(* Logix 5000 project; controller Sucrose_Main Emulate 5570 rev 20.12; software revision 20.01; part 10 of 30 *)
(* tags used below, declared in another part *)
   Alarm_ACK_Master_Timer : TIMER;
   DO_E20_6 : ALIAS FOR FLX_E20:6:O;   // Discrete Output EN2T_FLX 192.168.1.20
   DO_E20_7 : ALIAS FOR FLX_E20:7:O;   // Discrete Output EN2T_FLX 192.168.1.20
   DO_E24_3 : ALIAS FOR FLX_E24:3:O;   // Discrete Output EN2T_FLX 192.168.1.24
   FV230103_AOI : QSI_Flow_Valve;   // FV-23-01-03 SUCROSE TANK #1 OUTLET VALVE
   FV230203_AOI : QSI_Flow_Valve;   // FV-23-02-03 SUCROSE TANK #2 OUTLET VALVE
   FV230401_AOI : QSI_Flow_Valve;   // FV-23-04-01 SUCROSE TANK #3 LOW POINT DRAIN
   FV230402_AOI : QSI_Flow_Valve;   // FV-23-04-02 SUCROSE TANK #2 LOW POINT DRAIN
   FV230403_AOI : QSI_Flow_Valve;   // FV-23-04-03 SUCROSE TANK #1 LOW POINT DRAIN
   FV230431_AOI : QSI_Flow_Valve;   // FV-23-04-31 SUCROSE LOW POINT DRAIN VALVE @ TRANSFER PUMP #1
   FV230432_AOI : QSI_Flow_Valve;   // FV-23-04-32 SUCROSE LOW POINT DRAIN VALVE @ TRANSFER PUMP #2
   P230401_AOI : PF525_VFD_E_ENET;   // P-23-04-01 SUCROSE TRANSFER PUMP 1
   P230402_AOI : PF525_VFD_E_ENET;   // P-23-04-02 SUCROSE TRANSFER PUMP 2
   PSV230401_AOI : QSI_Flow_Valve;   // PSV-23-04-01 TRANSFER PUMP #1 BYPASS VALVE
   PSV230402_AOI : QSI_Flow_Valve;   // PSV-23-04-02 TRANSFER PUMP #2 BYPASS VALVE
   Sucrose_MM_Enable : BOOL;
   SucroseCIP_P230401_REMOTE : CIP_REMOTE;
   SucroseCIP_P230402_REMOTE : CIP_REMOTE;
   SucroseCIP_TK230101_REMOTE : CIP_REMOTE;
   SucroseCIP_TK230201_REMOTE : CIP_REMOTE;
   SucroseTanks : Area_Program;
   SV130401_AOI : QSI_Discrete_Device;   // SV-13-04-01 SUCROSE TRANSFER PUMP #1 SEAL WATER FLUSH VALVE
   SV130402_AOI : QSI_Discrete_Device;   // SV-13-04-02 SUCROSE TRANSFER PUMP #2 SEAL WATER FLUSH VALVE
(* DischargeArea_EN2T_IO_Discrete_DO_E20_5, continued *)

ROUTINE MainRoutine   (* ladder *)
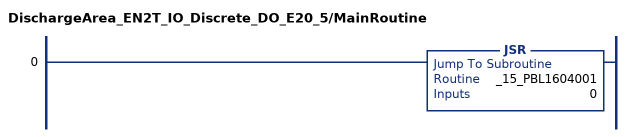
   0: JSR(_15_PBL1604001,0);
END_ROUTINE
END_PROGRAM

PROGRAM DischargeArea_EN2T_IO_Discrete_DO_E20_6   (* main routine MainRoutine *)

ROUTINE _00_FV230431   (* ladder *)
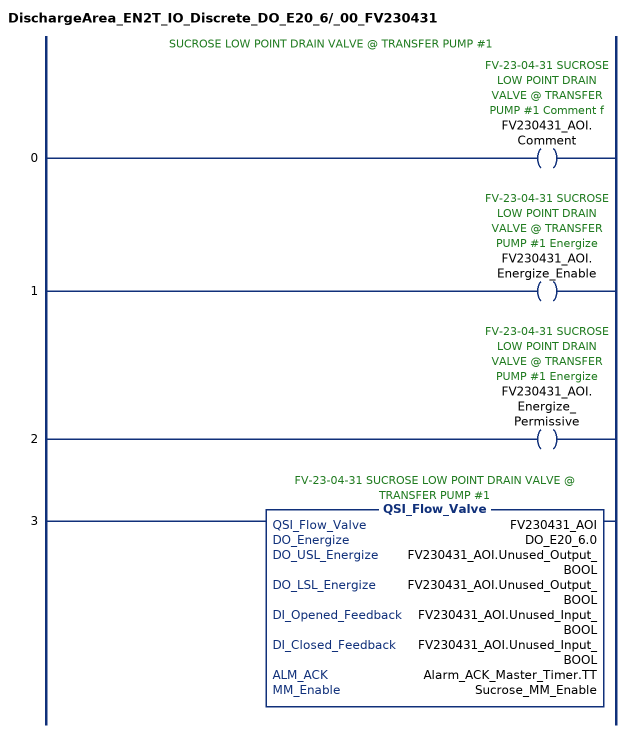
   // SUCROSE LOW POINT DRAIN VALVE @ TRANSFER PUMP #1
   0: OTE(FV230431_AOI.Comment);
   1: OTE(FV230431_AOI.Energize_Enable);
   2: OTE(FV230431_AOI.Energize_Permissive);
   3: QSI_Flow_Valve(FV230431_AOI,DO_E20_6.0,FV230431_AOI.Unused_Output_BOOL,FV230431_AOI.Unused_Output_BOOL,FV230431_AOI.Unused_Input_BOOL,FV230431_AOI.Unused_Input_BOOL,Alarm_ACK_Master_Timer.TT,Sucrose_MM_Enable);
END_ROUTINE

ROUTINE _01_FV230432   (* ladder *)
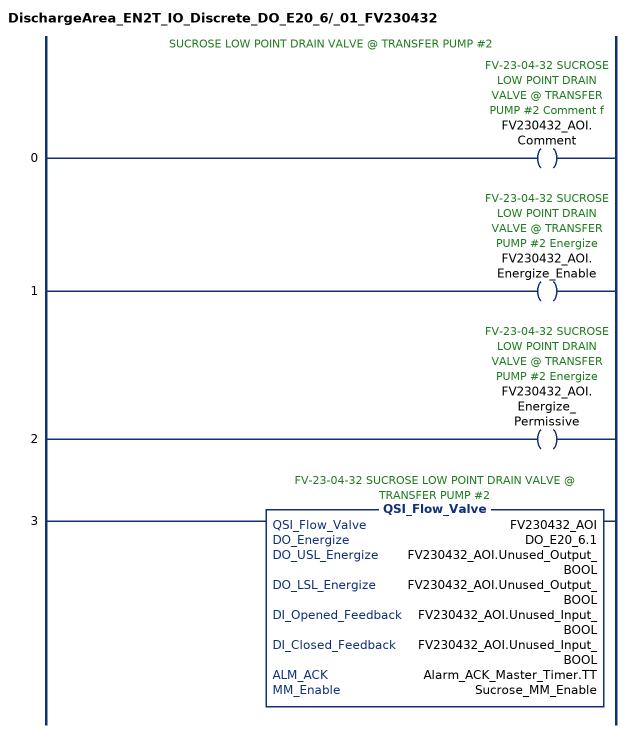
   // SUCROSE LOW POINT DRAIN VALVE @ TRANSFER PUMP #2
   0: OTE(FV230432_AOI.Comment);
   1: OTE(FV230432_AOI.Energize_Enable);
   2: OTE(FV230432_AOI.Energize_Permissive);
   3: QSI_Flow_Valve(FV230432_AOI,DO_E20_6.1,FV230432_AOI.Unused_Output_BOOL,FV230432_AOI.Unused_Output_BOOL,FV230432_AOI.Unused_Input_BOOL,FV230432_AOI.Unused_Input_BOOL,Alarm_ACK_Master_Timer.TT,Sucrose_MM_Enable);
END_ROUTINE

ROUTINE _04_FV230401   (* ladder *)
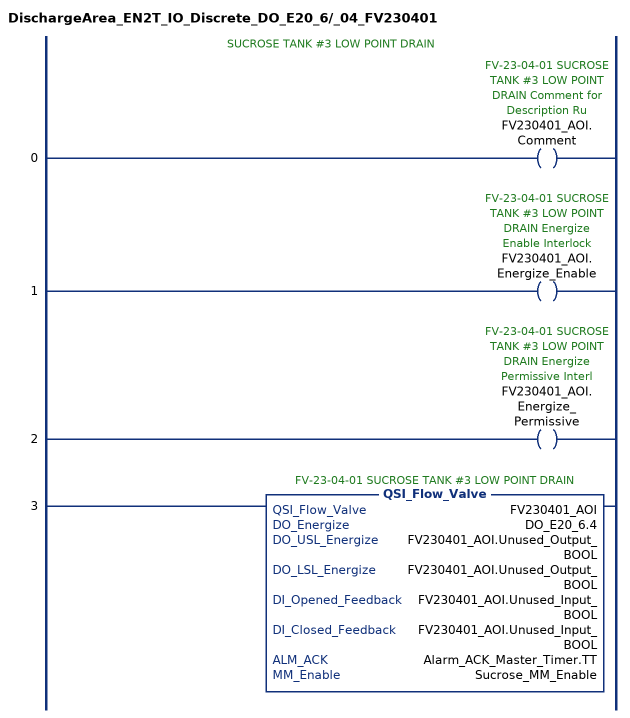
   // SUCROSE TANK #3 LOW POINT DRAIN
   0: OTE(FV230401_AOI.Comment);
   1: OTE(FV230401_AOI.Energize_Enable);
   2: OTE(FV230401_AOI.Energize_Permissive);
   3: QSI_Flow_Valve(FV230401_AOI,DO_E20_6.4,FV230401_AOI.Unused_Output_BOOL,FV230401_AOI.Unused_Output_BOOL,FV230401_AOI.Unused_Input_BOOL,FV230401_AOI.Unused_Input_BOOL,Alarm_ACK_Master_Timer.TT,Sucrose_MM_Enable);
END_ROUTINE

ROUTINE _05_FV230402   (* ladder *)
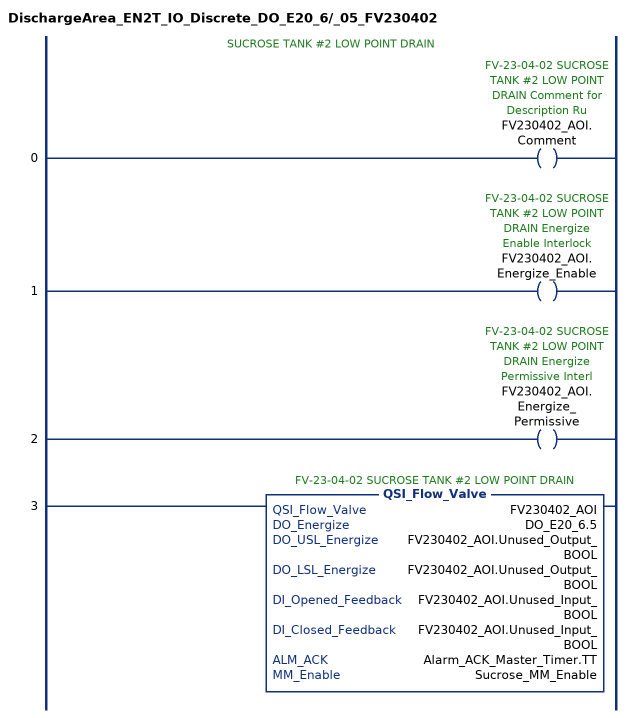
   // SUCROSE TANK #2 LOW POINT DRAIN
   0: OTE(FV230402_AOI.Comment);
   1: OTE(FV230402_AOI.Energize_Enable);
   2: OTE(FV230402_AOI.Energize_Permissive);
   3: QSI_Flow_Valve(FV230402_AOI,DO_E20_6.5,FV230402_AOI.Unused_Output_BOOL,FV230402_AOI.Unused_Output_BOOL,FV230402_AOI.Unused_Input_BOOL,FV230402_AOI.Unused_Input_BOOL,Alarm_ACK_Master_Timer.TT,Sucrose_MM_Enable);
END_ROUTINE

ROUTINE _06_FV230403   (* ladder *)
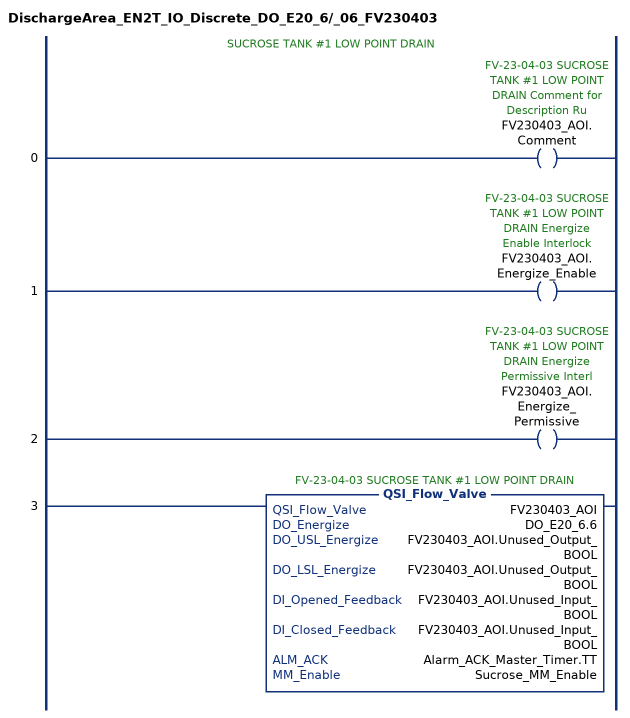
   // SUCROSE TANK #1 LOW POINT DRAIN
   0: OTE(FV230403_AOI.Comment);
   1: OTE(FV230403_AOI.Energize_Enable);
   2: OTE(FV230403_AOI.Energize_Permissive);
   3: QSI_Flow_Valve(FV230403_AOI,DO_E20_6.6,FV230403_AOI.Unused_Output_BOOL,FV230403_AOI.Unused_Output_BOOL,FV230403_AOI.Unused_Input_BOOL,FV230403_AOI.Unused_Input_BOOL,Alarm_ACK_Master_Timer.TT,Sucrose_MM_Enable);
END_ROUTINE

ROUTINE _08_PSV230401   (* ladder *)
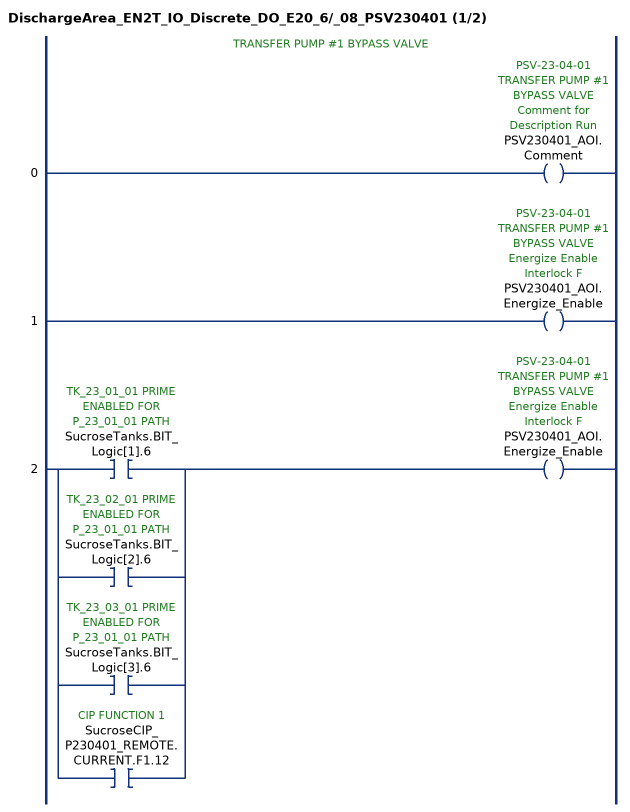
   // TRANSFER PUMP #1 BYPASS VALVE
   0: OTE(PSV230401_AOI.Comment);
   1: OTE(PSV230401_AOI.Energize_Enable);
   2: [XIC(SucroseTanks.BIT_Logic[1].6) ,XIC(SucroseTanks.BIT_Logic[2].6) ,XIC(SucroseTanks.BIT_Logic[3].6) ,XIC(SucroseCIP_P230401_REMOTE.CURRENT.F1.12) ]OTE(PSV230401_AOI.Energize_Enable);
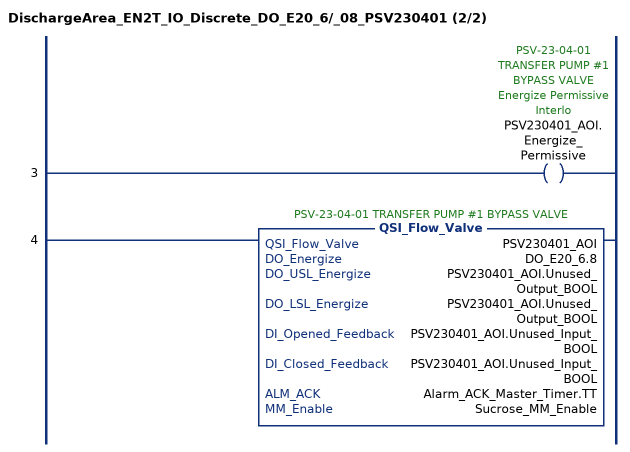
   3: OTE(PSV230401_AOI.Energize_Permissive);
   4: QSI_Flow_Valve(PSV230401_AOI,DO_E20_6.8,PSV230401_AOI.Unused_Output_BOOL,PSV230401_AOI.Unused_Output_BOOL,PSV230401_AOI.Unused_Input_BOOL,PSV230401_AOI.Unused_Input_BOOL,Alarm_ACK_Master_Timer.TT,Sucrose_MM_Enable);
END_ROUTINE

ROUTINE _09_PSV230402   (* ladder *)
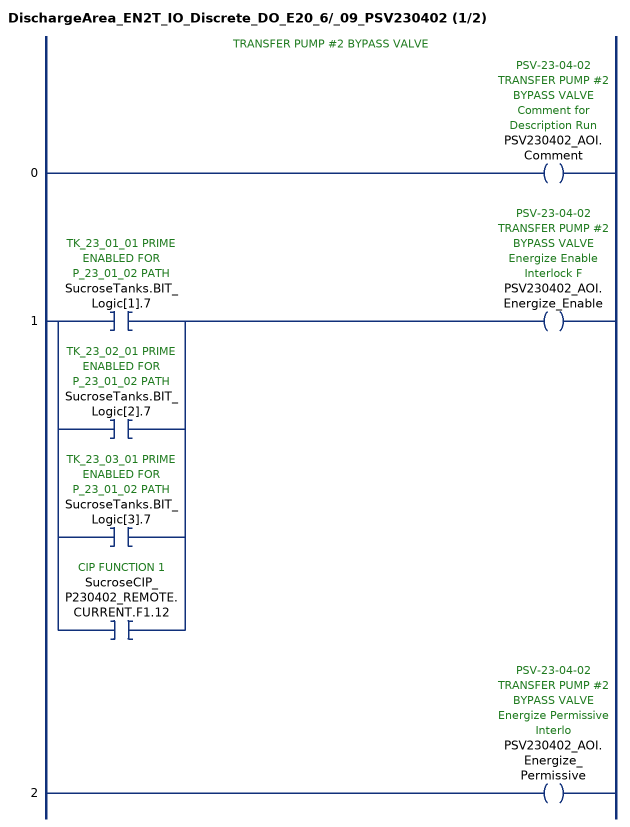
   // TRANSFER PUMP #2 BYPASS VALVE
   0: OTE(PSV230402_AOI.Comment);
   1: [XIC(SucroseTanks.BIT_Logic[1].7) ,XIC(SucroseTanks.BIT_Logic[2].7) ,XIC(SucroseTanks.BIT_Logic[3].7) ,XIC(SucroseCIP_P230402_REMOTE.CURRENT.F1.12) ]OTE(PSV230402_AOI.Energize_Enable);
   2: OTE(PSV230402_AOI.Energize_Permissive);
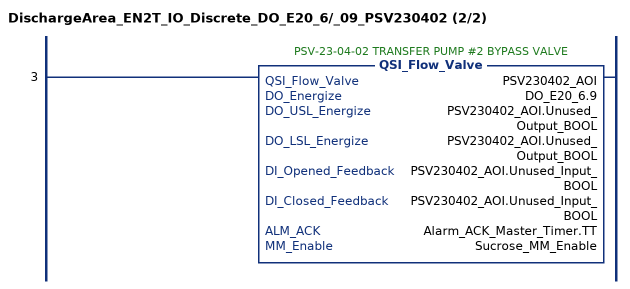
   3: QSI_Flow_Valve(PSV230402_AOI,DO_E20_6.9,PSV230402_AOI.Unused_Output_BOOL,PSV230402_AOI.Unused_Output_BOOL,PSV230402_AOI.Unused_Input_BOOL,PSV230402_AOI.Unused_Input_BOOL,Alarm_ACK_Master_Timer.TT,Sucrose_MM_Enable);
END_ROUTINE

ROUTINE MainRoutine   (* ladder *)
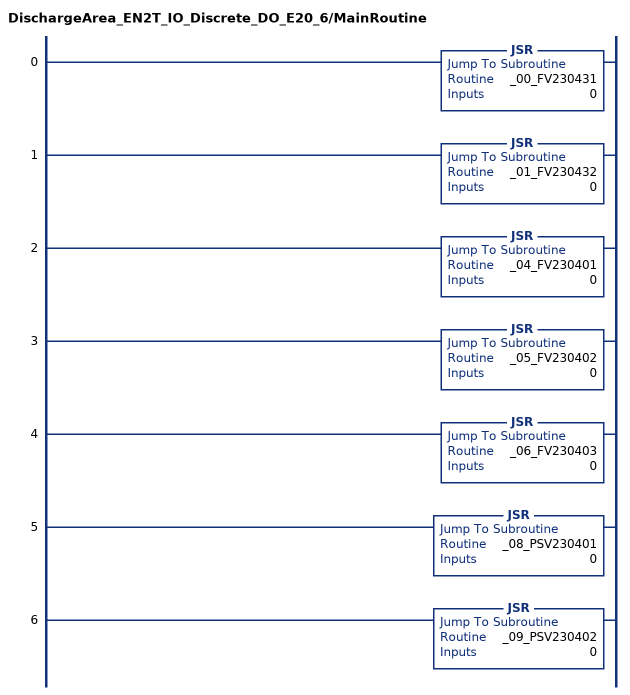
   0: JSR(_00_FV230431,0);
   1: JSR(_01_FV230432,0);
   2: JSR(_04_FV230401,0);
   3: JSR(_05_FV230402,0);
   4: JSR(_06_FV230403,0);
   5: JSR(_08_PSV230401,0);
   6: JSR(_09_PSV230402,0);
END_ROUTINE
END_PROGRAM

PROGRAM DischargeArea_EN2T_IO_Discrete_DO_E20_7   (* main routine MainRoutine *)

ROUTINE _00_SV130401   (* ladder *)
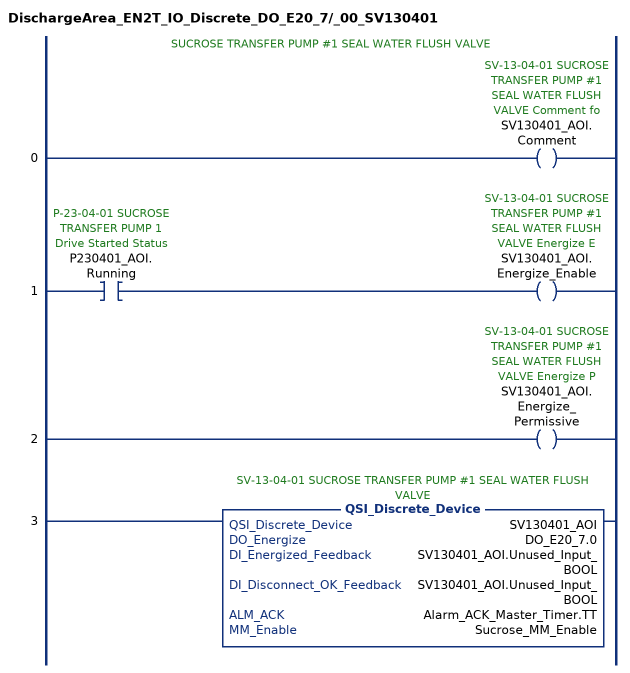
   // SUCROSE TRANSFER PUMP #1 SEAL WATER FLUSH VALVE
   0: OTE(SV130401_AOI.Comment);
   1: XIC(P230401_AOI.Running)OTE(SV130401_AOI.Energize_Enable);
   2: OTE(SV130401_AOI.Energize_Permissive);
   3: QSI_Discrete_Device(SV130401_AOI,DO_E20_7.0,SV130401_AOI.Unused_Input_BOOL,SV130401_AOI.Unused_Input_BOOL,Alarm_ACK_Master_Timer.TT,Sucrose_MM_Enable);
END_ROUTINE

ROUTINE _01_SV130402   (* ladder *)
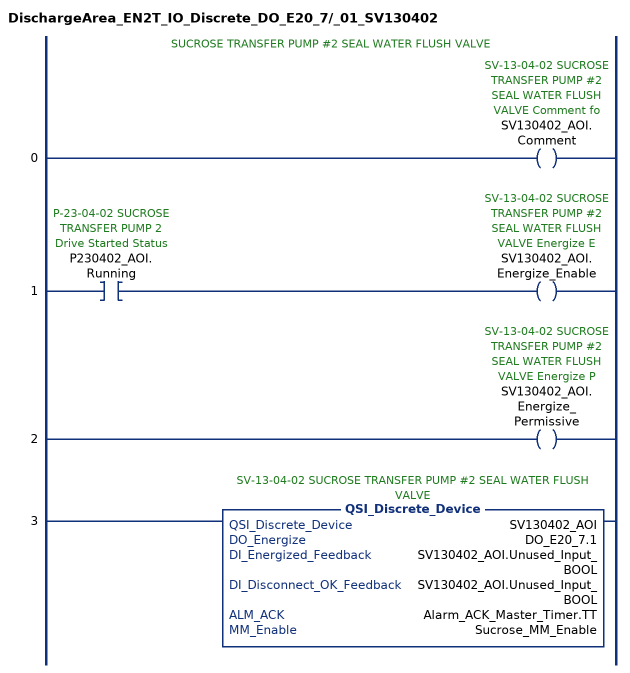
   // SUCROSE TRANSFER PUMP #2 SEAL WATER FLUSH VALVE
   0: OTE(SV130402_AOI.Comment);
   1: XIC(P230402_AOI.Running)OTE(SV130402_AOI.Energize_Enable);
   2: OTE(SV130402_AOI.Energize_Permissive);
   3: QSI_Discrete_Device(SV130402_AOI,DO_E20_7.1,SV130402_AOI.Unused_Input_BOOL,SV130402_AOI.Unused_Input_BOOL,Alarm_ACK_Master_Timer.TT,Sucrose_MM_Enable);
END_ROUTINE

ROUTINE MainRoutine   (* ladder *)
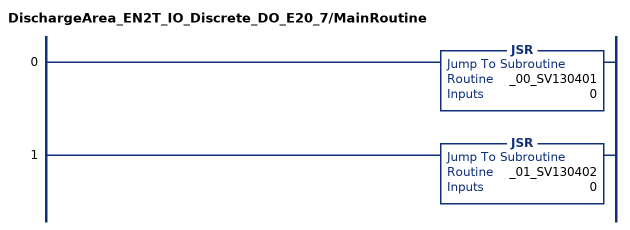
   0: JSR(_00_SV130401,0);
   1: JSR(_01_SV130402,0);
END_ROUTINE
END_PROGRAM

PROGRAM DischargeArea_EN2T_IO_Discrete_DO_E24_3   (* main routine MainRoutine *)

ROUTINE _01_FV230103   (* ladder *)
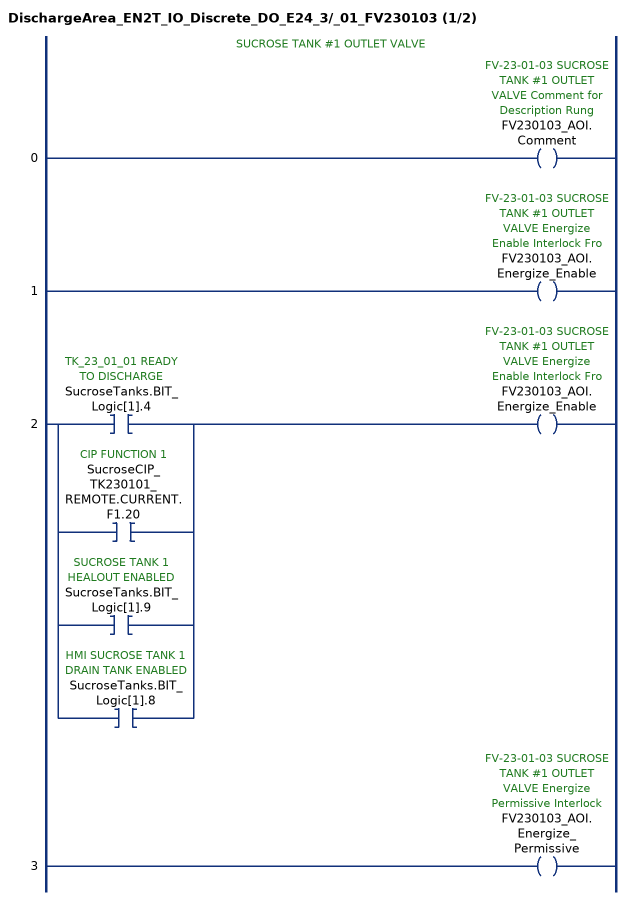
   // SUCROSE TANK #1 OUTLET VALVE
   0: OTE(FV230103_AOI.Comment);
   1: OTE(FV230103_AOI.Energize_Enable);
   2: [XIC(SucroseTanks.BIT_Logic[1].4) ,XIC(SucroseCIP_TK230101_REMOTE.CURRENT.F1.20) ,XIC(SucroseTanks.BIT_Logic[1].9) ,XIC(SucroseTanks.BIT_Logic[1].8) ]OTE(FV230103_AOI.Energize_Enable);
   3: OTE(FV230103_AOI.Energize_Permissive);
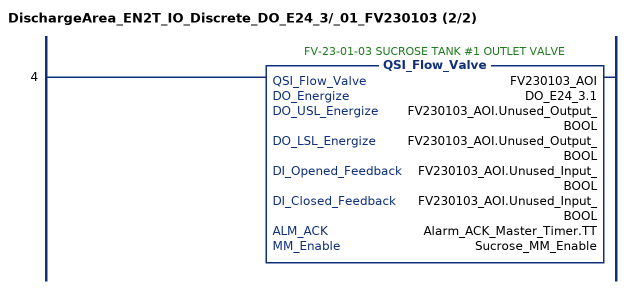
   4: QSI_Flow_Valve(FV230103_AOI,DO_E24_3.1,FV230103_AOI.Unused_Output_BOOL,FV230103_AOI.Unused_Output_BOOL,FV230103_AOI.Unused_Input_BOOL,FV230103_AOI.Unused_Input_BOOL,Alarm_ACK_Master_Timer.TT,Sucrose_MM_Enable);
END_ROUTINE

ROUTINE _05_FV230203   (* ladder *)
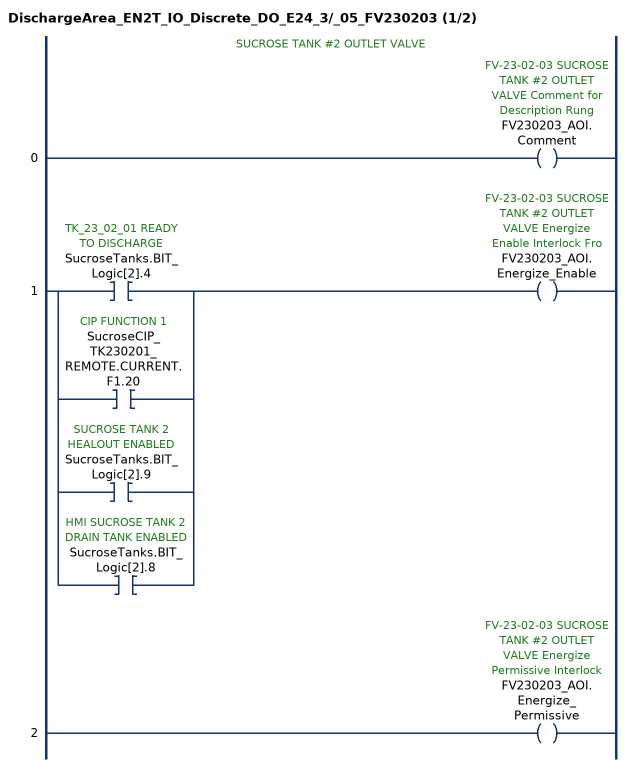
   // SUCROSE TANK #2 OUTLET VALVE
   0: OTE(FV230203_AOI.Comment);
   1: [XIC(SucroseTanks.BIT_Logic[2].4) ,XIC(SucroseCIP_TK230201_REMOTE.CURRENT.F1.20) ,XIC(SucroseTanks.BIT_Logic[2].9) ,XIC(SucroseTanks.BIT_Logic[2].8) ]OTE(FV230203_AOI.Energize_Enable);
   2: OTE(FV230203_AOI.Energize_Permissive);
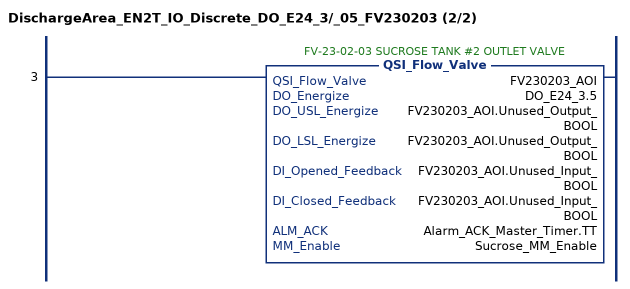
   3: QSI_Flow_Valve(FV230203_AOI,DO_E24_3.5,FV230203_AOI.Unused_Output_BOOL,FV230203_AOI.Unused_Output_BOOL,FV230203_AOI.Unused_Input_BOOL,FV230203_AOI.Unused_Input_BOOL,Alarm_ACK_Master_Timer.TT,Sucrose_MM_Enable);
END_ROUTINE
